SUBAPPLICATION Uebung_012h_AR2 (* Nur OPC-UA (kein VT-Feld) und Speichern NVS via AR2 - OPC_TO_AR2 direkt an ein NVS_AR2 angeschlossen *)
  (* Standard: 61499-2; Description: Copyright (c) 2026 Meisterschulen am Ostbahnhof This program and the accompanying materials are made available under the terms of the Eclipse Public License 2.0 which is available at https://www.eclipse.org/legal/epl-2.0/ SPDX-License-Identifier: EPL-2.0 *)
  (* Version 1.0, 2026-08-31, Franz Höpfinger, Meisterschulen am Ostbahnhof, OPC-only sibling of Uebung_012d_AR2 (VT only) - kein VT-Objekt, nur Remote-Subscribe/Publish via OPC_TO_AR2 direkt an NVS_AR2 *)
  PACKAGE Uebungen;
  IMPORT Uebungen::const::NVS::NVS_Keys::KEY_I1_STORE;
  IMPORT Uebungen::const::OPC::OPC_Strings::Uebung12h_READ;
  IMPORT Uebungen::const::OPC::OPC_Strings::Uebung12h_WRITE;
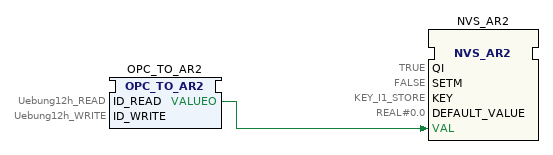
  (* Kein VT-Feld noetig - der Wert kommt ausschliesslich per OPC-UA. SETM=FALSE reicht hier: es gibt nur EINE Quelle (Remote), also keine 'andere Seite', die live ueber eine Aenderung informiert werden muesste. Der Boot-Wert laedt trotzdem immer korrekt (INIT->INITO->GET->GETO, unabhaengig von SETM). *)
  FBS
    NVS_AR2 : logiBUS::storage::esp32_nvs::NVS_AR2(QI := TRUE, SETM := FALSE, KEY := KEY_I1_STORE, DEFAULT_VALUE := REAL#0.0);
  END_FBS
  SUBAPPS
    OPC_TO_AR2 : MyLib::sys::OPC_TO_AR2(ID_READ := Uebung12h_READ, ID_WRITE := Uebung12h_WRITE);
  END_SUBAPPS
  ADAPTER_CONNECTIONS
    OPC_TO_AR2.VALUEO TO NVS_AR2.VAL;
  END_CONNECTIONS
END_SUBAPPLICATION
